(* IEC 61131-3 sources: netRob/Hardwareadapter/parser/misc/data, 6 files *)

(* ---- GeneralConstants.IEC ---- *)
TYPE GeneralConstants :
	STRUCT
		(* Constants *)
		KEY_SIZE: UINT;
		TEXT_VALUE_SIZE: UINT;
		MAX_NESTING_DEPTH: UINT;
	END_STRUCT
END_TYPE

(* ---- NestedKeys.IEC ---- *)
TYPE NestedKeys :
	ARRAY[1..10] OF JsonKey; (* 10 <=> Constants.MAX_NESTING_DEPTH *)
END_TYPE

(* ---- STRING1.IEC ---- *)
TYPE STRING1 :
	STRING(1);
END_TYPE

(* ---- StringKeySize.IEC ---- *)
TYPE StringKeySize :
	STRING(255); (* STRING(Constants_KEY_SIZE) *)
END_TYPE

(* ---- StringTextSize.IEC ---- *)
TYPE StringTextSize :
	STRING(1024); (* STRING(Constants_TEXT_VALUE_SIZE) *)
END_TYPE

(* ---- ParserGlobals.IEC ---- *)
VAR_GLOBAL
	Constants: GeneralConstants;
	resetParser: BOOL := FALSE;
END_VAR
